DATA_BLOCK "MotorControl"
{ S7_Optimized_Access := 'TRUE' }
VERSION : 0.1
NON_RETAIN
   VAR
      Dev { S7_SetPoint := 'False'} : Array[1..20] of "Motor_Control";
   END_VAR


BEGIN

END_DATA_BLOCK

